Yaskawa INFORM job: X2_54(90,90).JBI

/JOB
//NAME X2_54(90,90)
//POS
///NPOS 83,83,83,5,0,0
///TOOL 0
///POSTYPE PULSE
///PULSE
C00000=-1588,-95931,-85547,536,91020,79
C00001=109614,-80770,-33274,-26441,88313,59950
C00002=123848,-31777,-18455,-23445,107090,61187
C00003=123841,-28849,-10488,-23011,103953,61824
C00004=121631,-31502,-9740,-23500,101656,61457
C00005=120611,-52731,-25618,-22979,88766,63590
C00006=120611,-52127,-24298,-22979,88302,63679
C00007=120709,-31590,-7271,-23636,99957,61459
C00008=120709,-31590,-7271,-23636,99957,61459
C00009=119091,-31571,-7259,-24123,99501,60955
C00010=120709,-31590,-7271,-23636,99957,61459
C00011=120709,-32483,-9368,-23711,100721,61304
C00012=120710,-25083,-4381,-23781,101396,61167
C00013=121006,-24761,-1298,-23531,99887,61582
C00014=121017,-27452,-3154,-23507,99669,61631
C00015=121006,-24761,-1298,-23531,99887,61582
C00016=123867,-28847,-10487,-23003,103961,61832
C00017=133172,-25083,-9106,-11800,111088,-60653
C00018=133980,-32103,-11521,-11286,109122,-60157
C00019=134476,-34965,-10517,-10928,107138,-59789
C00020=134477,-34405,-9236,-10895,106647,-59744
C00021=134476,-35484,-11718,-10961,107602,-59833
C00022=133816,-29381,-7710,-11281,108171,-60124
C00023=133893,-26907,-1983,-11094,105969,-59888
C00024=134173,-29539,-3766,-10963,105756,-59769
C00025=133893,-26907,-1983,-11094,105969,-59888
C00026=133172,-25083,-9106,-11800,111088,-60653
C00027=121137,-36213,-21218,-16738,109595,-64926
C00028=120773,-142410,-68657,-16722,68160,-59618
C00029=120750,-136737,-62500,-16824,67318,-59502
C00030=120694,-76236,-37859,-16915,92835,-62927
C00031=120643,-40052,-18916,-16620,107300,-64838
C00032=120644,-37132,-13487,-16440,105532,-64588
C00033=120748,-35212,-10478,-16324,104724,-64435
C00034=120672,-34760,-9448,-16318,104322,-64407
C00035=120672,-35841,-11929,-16403,105256,-64537
C00036=120662,-29717,-7920,-16469,105906,-64632
C00037=120661,-27286,-2266,-16274,103763,-64334
C00038=120665,-29958,-4070,-16251,103510,-64298
C00039=120661,-27286,-2266,-16274,103763,-64334
C00040=120652,-25328,-9262,-16793,108862,-65060
C00041=123773,-22568,-7529,17624,103248,-64219
C00042=124327,-26442,-6307,17576,100510,-64424
C00043=126313,-25888,-5320,18125,99773,-63823
C00044=126313,-25209,-3680,18082,99144,-63918
C00045=126313,-26231,-6162,18148,100099,-63774
C00046=122777,-47933,-21609,20152,87002,-62388
C00047=124588,-47820,-21545,20396,86579,-61819
C00048=122777,-47933,-21609,20152,87002,-62388
C00049=122777,-48866,-23702,20148,87762,-62262
C00050=114705,-22863,1172,28112,98540,-64375
C00051=114366,-20787,5741,27869,97101,-64853
C00052=114243,-23463,3841,27816,96957,-64934
C00053=114366,-20787,5741,27869,97101,-64853
C00054=111202,-25367,-3960,27262,101348,-65029
C00055=95937,-14786,-4111,12325,115184,58222
C00056=95439,-18182,-3602,11879,113244,57819
C00057=95226,-19598,-3618,11714,112572,57667
C00058=143581,-21076,-4592,28938,100124,73729
C00059=134161,-30122,-6272,39681,94062,72864
C00060=122849,-36840,-3636,50267,89979,70728
C00061=120332,-34990,-5150,49750,92548,70847
C00062=111071,-38110,-13453,47846,99778,69985
C00063=98656,-103112,-42086,41787,94311,61961
C00064=120779,-143878,-70215,-16699,68357,-59644
C00065=121136,-35849,-20201,-16687,109174,-64865
C00066=140438,-19542,-8678,1398,106615,-76287
C00067=140798,-23007,-8136,1496,104495,-76185
C00068=140939,-24203,-7667,1533,103589,-76150
C00069=100286,-20336,-2562,-22406,99032,-78449
C00070=110627,-28233,-3813,-33814,93632,-77860
C00071=122197,-34580,-2434,-43859,90621,-76172
C00072=124529,-32488,-3757,-43384,93122,-76205
C00073=128873,-21855,-1396,-42713,98174,-76387
C00074=122911,-31943,-14008,19509,93775,-82296
C00075=116294,-42254,-22825,16168,95841,-83791
C00076=116243,-43675,-23679,16151,95655,-83834
C00077=115646,-43881,-22062,15991,94710,-84166
C00078=157537,-25683,-3175,37597,77487,-74154
C00079=138669,-32638,-13170,36057,87562,-78565
C00080=117127,-39145,-23396,32899,98704,-83849
C00081=84432,-67942,-39671,-7809,93678,-73867
C00082=-1588,-95931,-85547,536,91020,79
BC00000=197629,523905,680388
BC00001=296350,518660,473051
BC00002=330153,435557,392508
BC00003=330153,435557,392508
BC00004=330153,435557,392508
BC00005=330153,435557,392508
BC00006=330153,435557,392508
BC00007=330153,435557,392508
BC00008=330153,435557,392508
BC00009=330153,435557,392508
BC00010=330153,435557,392508
BC00011=330153,435557,392508
BC00012=330153,435557,392508
BC00013=330153,435557,392508
BC00014=330153,435557,392508
BC00015=330153,435557,392508
BC00016=330153,435557,392508
BC00017=274759,420582,401695
BC00018=274759,420582,401695
BC00019=274759,420582,401695
BC00020=274759,420582,401695
BC00021=274759,420582,401695
BC00022=274759,420582,401695
BC00023=274759,420582,401695
BC00024=274759,420582,401695
BC00025=274759,420582,401695
BC00026=274759,420582,401695
BC00027=289302,420692,401698
BC00028=304429,422463,401752
BC00029=98759,422463,401752
BC00030=101123,398567,401752
BC00031=138754,413503,401752
BC00032=139894,422463,401752
BC00033=139894,422463,401752
BC00034=139894,422463,401752
BC00035=139894,422463,401752
BC00036=139894,422463,401752
BC00037=139894,422463,401752
BC00038=139894,422463,401752
BC00039=139894,422463,401752
BC00040=139894,422463,401752
BC00041=105393,442576,405335
BC00042=105393,442576,405335
BC00043=105393,442576,405335
BC00044=105393,442576,405335
BC00045=105393,442576,405335
BC00046=105393,442576,405335
BC00047=105393,442576,405335
BC00048=105393,442576,405335
BC00049=105393,442576,405335
BC00050=105393,442576,405335
BC00051=105393,442576,405335
BC00052=105393,442576,405335
BC00053=105393,442576,405335
BC00054=105393,442576,405335
BC00055=143733,432604,364759
BC00056=143733,432604,364759
BC00057=143733,432604,364759
BC00058=143733,432604,364759
BC00059=143733,432604,364759
BC00060=143733,432604,364759
BC00061=143733,432604,364759
BC00062=143733,432604,364759
BC00063=143733,432604,364759
BC00064=304429,422463,401752
BC00065=289302,420692,401698
BC00066=306452,436520,388561
BC00067=306452,436520,388561
BC00068=306452,436520,388561
BC00069=306452,436520,388561
BC00070=306452,436520,388561
BC00071=306452,436520,388561
BC00072=306452,436520,388561
BC00073=306452,436520,388561
BC00074=306452,436520,388561
BC00075=296471,435362,388593
BC00076=296471,435362,388593
BC00077=296471,435362,388593
BC00078=296471,435362,388593
BC00079=296471,435362,388593
BC00080=296471,435362,388593
BC00081=227708,523893,389113
BC00082=197629,523905,680388
EC00000=-798156,-740307
EC00001=-798156,-740307
EC00002=-798156,-740307
EC00003=-798156,-740307
EC00004=-798156,-740307
EC00005=-798156,-740307
EC00006=-798156,-740307
EC00007=-798156,-740307
EC00008=-798156,-740307
EC00009=-798156,-740307
EC00010=-798156,-740307
EC00011=-798156,-740307
EC00012=-798156,-740307
EC00013=-798156,-740307
EC00014=-798156,-740307
EC00015=-798156,-740307
EC00016=-798156,-740307
EC00017=-798156,-740307
EC00018=-798156,-740307
EC00019=-798156,-740307
EC00020=-798156,-740307
EC00021=-798156,-740307
EC00022=-798156,-740307
EC00023=-798156,-740307
EC00024=-798156,-740307
EC00025=-798156,-740307
EC00026=-798156,-740307
EC00027=-798156,-740307
EC00028=-798156,-740307
EC00029=-798156,-740307
EC00030=-798156,-740307
EC00031=-798156,-740307
EC00032=-798156,-740307
EC00033=-798156,-740307
EC00034=-798156,-740307
EC00035=-798156,-740307
EC00036=-798156,-740307
EC00037=-798156,-740307
EC00038=-798156,-740307
EC00039=-798156,-740307
EC00040=-798156,-740307
EC00041=-798156,-740307
EC00042=-798156,-740307
EC00043=-798156,-740307
EC00044=-798156,-740307
EC00045=-798156,-740307
EC00046=-798156,-740307
EC00047=-798156,-740307
EC00048=-798156,-740307
EC00049=-798156,-740307
EC00050=-798156,-740307
EC00051=-798156,-740307
EC00052=-798156,-740307
EC00053=-798156,-740307
EC00054=-798156,-740307
EC00055=-798156,-740307
EC00056=-798156,-740307
EC00057=-798156,-740307
EC00058=-798156,-740307
EC00059=-798156,-740307
EC00060=-798156,-740307
EC00061=-798156,-740307
EC00062=-798156,-740307
EC00063=-798156,-740307
EC00064=-798156,-740307
EC00065=-798156,-740307
EC00066=-798156,-740307
EC00067=-798156,-740307
EC00068=-798156,-740307
EC00069=-798156,-740307
EC00070=-798156,-740307
EC00071=-798156,-740307
EC00072=-798156,-740307
EC00073=-798156,-740307
EC00074=-798156,-740307
EC00075=-798156,-740307
EC00076=-798156,-740307
EC00077=-798156,-740307
EC00078=-798156,-740307
EC00079=-798156,-740307
EC00080=-798156,-740307
EC00081=-798156,-740307
EC00082=-798156,-740307
///POSTYPE BASE
///RECTAN
///RCONF 0,0,0,0,1,0,0,0,0,0,0,0,0,0,0,0,0,0,0,0,0,0,0,0
P00006=2.006,1.622,-0.565,0.0000,0.0000,0.0000
P00021=0.073,2.058,-0.109,0.0000,0.0000,0.0000
P00022=2.006,1.622,-0.565,0.0000,0.0000,0.0000
///RCONF 0,0,0,0,0,0,0,0,0,0,0,0,0,0,0,0,0,0,0,0,0,0,0,0
P00023=-2.957,-4.083,2.762,0.0000,0.0000,0.0000
P00024=-1.466,-0.226,-0.419,0.0000,0.0000,0.0000
//INST
///DATE 2024/12/10 19:29
///ATTR SC,RW
///GROUP1 RB1,BS1
///GROUP2 ST1
NOP
'X2_54(90,90)
MOVJ C00000 BC00000 VJ=100.00  +MOVJ EC00000 VJ=100.00
MOVJ C00001 BC00001 VJ=100.00  +MOVJ EC00001 VJ=100.00
MOVJ C00002 BC00002 VJ=100.00  +MOVJ EC00002 VJ=100.00
'Path S3753
SFTOF3D
MOVJ C00003 BC00003 VJ=100.00  +MOVJ EC00003 VJ=100.00
MOVL C00004 BC00004 V=666.7  +MOVJ EC00004 VJ=100.00
SMOVL C00005 BC00005 V=166.7  +MOVJ EC00005
SREFP 3 C00006 BC00006  +REFP EC00006
CALL JOB:SEARCH-R1-S13D
SET P021 P006
SFTON3D P021
SMOVL C00007 BC00007 V=166.7  +MOVJ EC00007
SMOVL C00008 BC00008 V=166.7  +MOVJ EC00008
SREFP 3 C00009 BC00009  +REFP EC00009
CALL JOB:SEARCH-R1-S13D
SET P021 P006
SFTON3D P021
SMOVL C00010 BC00010 V=166.7  +MOVJ EC00010
SMOVL C00011 BC00011 V=333.3  +MOVJ EC00011
SMOVL C00012 BC00012 V=333.3  +MOVJ EC00012
SMOVL C00013 BC00013 V=250.0  +MOVJ EC00013
SREFP 3 C00014 BC00014  +REFP EC00014
CALL JOB:SEARCH-R1-S13D
SET P021 P006
SFTON3D P021
SMOVL C00015 BC00015 V=166.7  +MOVJ EC00015
MOVL C00016 BC00016 V=1000.0  +MOVJ EC00016 VJ=100.00
'EndPath S3753
'Path S3752
SFTOF3D
MOVJ C00017 BC00017 VJ=100.00  +MOVJ EC00017 VJ=100.00
SMOVL C00018 BC00018 V=666.7  +MOVJ EC00018
SMOVL C00019 BC00019 V=166.7  +MOVJ EC00019
SREFP 3 C00020 BC00020  +REFP EC00020
CALL JOB:SEARCH-R1-S13D
SET P022 P006
SFTON3D P022
SMOVL C00021 BC00021 V=800.0  +MOVJ EC00021
SMOVL C00022 BC00022 V=800.0  +MOVJ EC00022
SMOVL C00023 BC00023 V=200.0  +MOVJ EC00023
SREFP 3 C00024 BC00024  +REFP EC00024
CALL JOB:SEARCH-R1-S13D
SET P022 P006
SFTON3D P022
SMOVL C00025 BC00025 V=166.7  +MOVJ EC00025
MOVL C00026 BC00026 V=1000.0  +MOVJ EC00026 VJ=100.00
'EndPath S3752
MOVJ C00027 BC00027 VJ=100.00  +MOVJ EC00027 VJ=100.00
MOVJ C00028 BC00028 VJ=100.00  +MOVJ EC00028 VJ=100.00
MOVJ C00029 BC00029 VJ=100.00  +MOVJ EC00029 VJ=100.00
'Path S4334
SFTOF3D
MOVJ C00030 BC00030 VJ=20.00  +MOVJ EC00030 VJ=20.00
MOVJ C00031 BC00031 VJ=100.00  +MOVJ EC00031 VJ=100.00
MOVL C00032 BC00032 V=800.0  +MOVJ EC00032 VJ=100.00
SMOVL C00033 BC00033 V=166.7  +MOVJ EC00033
SREFP 3 C00034 BC00034  +REFP EC00034
CALL JOB:SEARCH-R1-S13D
SET P023 P006
SFTON3D P023
SMOVL C00035 BC00035 V=250.0  +MOVJ EC00035
SMOVL C00036 BC00036 V=250.0  +MOVJ EC00036
SMOVL C00037 BC00037 V=200.0  +MOVJ EC00037
SREFP 3 C00038 BC00038  +REFP EC00038
CALL JOB:SEARCH-R1-S13D
SET P023 P006
SFTON3D P023
SMOVL C00039 BC00039 V=250.0  +MOVJ EC00039
MOVL C00040 BC00040 V=1000.0  +MOVJ EC00040 VJ=100.00
'EndPath S4334
'Path S3751
SFTOF3D
MOVJ C00041 BC00041 VJ=100.00  +MOVJ EC00041 VJ=100.00
SMOVL C00042 BC00042 V=666.7  +MOVJ EC00042
SMOVL C00043 BC00043 V=166.7  +MOVJ EC00043
SREFP 3 C00044 BC00044  +REFP EC00044
CALL JOB:SEARCH-R1-S13D
SET P024 P006
SFTON3D P024
SMOVL C00045 BC00045 V=250.0  +MOVJ EC00045
SMOVL C00046 BC00046 V=166.7  +MOVJ EC00046
SREFP 3 C00047 BC00047  +REFP EC00047
CALL JOB:SEARCH-R1-S13D
SET P024 P006
SFTON3D P024
SMOVL C00048 BC00048 V=166.7  +MOVJ EC00048
SMOVL C00049 BC00049 V=250.0  +MOVJ EC00049
SMOVL C00050 BC00050 V=250.0  +MOVJ EC00050
SMOVL C00051 BC00051 V=250.0  +MOVJ EC00051
SREFP 3 C00052 BC00052  +REFP EC00052
CALL JOB:SEARCH-R1-S13D
SET P024 P006
SFTON3D P024
SMOVL C00053 BC00053 V=166.7  +MOVJ EC00053
MOVL C00054 BC00054 V=1000.0  +MOVJ EC00054 VJ=100.00
'EndPath S3751
'Path W4332
SFTOF3D
SFTON3D P023
MOVJ C00055 BC00055 VJ=100.00  +MOVJ EC00055 VJ=100.00
SMOVL C00056 BC00056 V=800.0  +MOVJ EC00056
SMOVL C00057 BC00057 V=150.0 PL=0  +MOVJ EC00057
MACRO1 MJ#(0) ARGF9
ARCON
SFTON3D P024
SMOVL C00058 BC00058 V=11.7  +MOVJ EC00058
SFTON3D P024
SMOVL C00059 BC00059 V=11.7  +MOVJ EC00059
ARCOF
SMOVL C00060 BC00060 V=800.0  +MOVJ EC00060
SMOVL C00061 BC00061 V=1000.0  +MOVJ EC00061
SFTOF3D
'EndPath W4332
MOVJ C00062 BC00062 VJ=100.00  +MOVJ EC00062 VJ=100.00
MOVJ C00063 BC00063 VJ=100.00  +MOVJ EC00063 VJ=100.00
MOVJ C00064 BC00064 VJ=100.00  +MOVJ EC00064 VJ=100.00
MOVJ C00065 BC00065 VJ=100.00  +MOVJ EC00065 VJ=100.00
'Path W4334
SFTOF3D
SFTON3D P022
MOVJ C00066 BC00066 VJ=100.00  +MOVJ EC00066 VJ=100.00
SMOVL C00067 BC00067 V=800.0  +MOVJ EC00067
SMOVL C00068 BC00068 V=150.0 PL=0  +MOVJ EC00068
ARCON
SFTON3D P021
SMOVL C00069 BC00069 V=11.7  +MOVJ EC00069
SFTON3D P021
SMOVL C00070 BC00070 V=11.7  +MOVJ EC00070
ARCOF
SMOVL C00071 BC00071 V=800.0  +MOVJ EC00071
SMOVL C00072 BC00072 V=1000.0  +MOVJ EC00072
SFTOF3D
'EndPath W4334
MOVJ C00073 BC00073 VJ=100.00  +MOVJ EC00073 VJ=100.00
MOVJ C00074 BC00074 VJ=100.00  +MOVJ EC00074 VJ=100.00
'Path W4333
SFTOF3D
SFTON3D P022
MOVJ C00075 BC00075 VJ=100.00  +MOVJ EC00075 VJ=100.00
SMOVL C00076 BC00076 V=800.0  +MOVJ EC00076
SMOVL C00077 BC00077 V=150.0 PL=0  +MOVJ EC00077
ARCON
SFTON3D P023
SMOVL C00078 BC00078 V=11.7  +MOVJ EC00078
ARCOF
SMOVL C00079 BC00079 V=800.0  +MOVJ EC00079
SMOVL C00080 BC00080 V=1000.0  +MOVJ EC00080
SFTOF3D
'EndPath W4333
MOVJ C00081 BC00081 VJ=50.00  +MOVJ EC00081 VJ=100.00
MOVJ C00082 BC00082 VJ=100.00  +MOVJ EC00082 VJ=100.00
END
